{attribute 'GeneratedUsingTerminal: EL7332-0000-0024'}
{attribute addProperty BoxType "EL7332-0000-0024"}
{attribute addProperty Id "StatusAT %I*Status_B679584511"}
{attribute addProperty CRC "921504111"}
{attribute addProperty Size "11"}
TYPE DCM_Status_Channel_36ED096F EXTENDS TcoIo.InputBase_8311D824 :
STRUCT
	{attribute addProperty Name "Status"}
	Status AT %I* : Status_B6795845;
END_STRUCT
END_TYPE

(* stored: Version 1.2.0.0, ProductVersion 3.1.4024.11
   DUT DCM_Status_Channel_36ED096F: Id {bb23b0c8-f5d5-05a4-06d6-8aee01c26078} *)
